{attribute addProperty BoxType "EK1100-0000-0018"}
{attribute addProperty Id "Beckhoff_APS1xxxEK1122Beckhoff_APS1xxxEK1122_5C62C20C2128266A_0002_APS1003_5000_0016APS1003_147A86932560320"}
{attribute addProperty CRC "1012690527"}
{attribute addProperty SizeInBites "4688"}
{attribute addProperty SizeInBytes "586"}
TYPE Beckhoff_APS1xxx_3C5C6E5F EXTENDS EK1100_179A0949 :
STRUCT
	{attribute addProperty Name "Beckhoff_APS1xxxEK1122"}
	Beckhoff_APS1xxxEK1122 : Beckhoff_APS1xxxEK1122_5C62C20C;
	{attribute addProperty Name "A_0002_APS1003_5000_0016"}
	A_0002_APS1003_5000_0016 : APS1003_147A8693;
END_STRUCT
END_TYPE

(* stored: Version 1.2.0.0, ProductVersion 3.1.4024.9
   DUT Beckhoff_APS1xxx_3C5C6E5F: Id {0145344a-eec7-414a-9ef5-3d23872a4288} *)
